// TIA Portal V20 export
TYPE "LER_typeHipotTrackingData"
// stored: Access Published
   STRUCT
      finished { ExternalWritable := 'False'} : Bool;
      result { ExternalWritable := 'False'} : Bool;
      data { ExternalWritable := 'False'} : String[26];
   END_STRUCT;
END_TYPE
